TYPE st_TCME31_Set_1 :
STRUCT
	IPAddress		:	String := '192.168.1.70';
	
	DigitalOutput1	:	Bool;
	DigitalOutput2	:	Bool;
	DigitalOutput3	:	Bool;
	DigitalOutput4	:	Bool;
END_STRUCT
END_TYPE

(* stored: Version 1.1.0.1, ProductVersion 3.1.4026.18
   DUT st_TCME31_Set_1: Id {4574e834-4668-47df-9d15-0fdca8d95a07} *)
